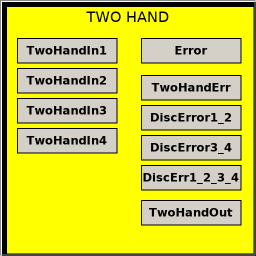
VISUALIZATION V_PH_TWOHAND  // 256x256
VAR_INPUT
	stSafetyTWOHAND			:ST_SAFETY_FBTWOHAND;
END_VAR
    Rectangle (2,2 256x256), colour toggle: stSafetyTWOHAND.bGeneralError
    Label (5,6 246x22), "TWO HAND"
    RoundedRectangle (17,38 100x25), "TwoHandIn1", colour toggle: stSafetyTWOHAND.uStatus.stStatusWords.wInputs.8
    RoundedRectangle (17,98 100x25), "TwoHandIn3", colour toggle: stSafetyTWOHAND.uStatus.stStatusWords.wInputs.10
    RoundedRectangle (17,68 100x25), "TwoHandIn2", colour toggle: stSafetyTWOHAND.uStatus.stStatusWords.wInputs.9
    RoundedRectangle (17,128 100x25), "TwoHandIn4", colour toggle: stSafetyTWOHAND.uStatus.stStatusWords.wInputs.11
    RoundedRectangle (141,38 100x25), "Error", colour toggle: stSafetyTWOHAND.uStatus.stStatusWords.wOutputs.0
    RoundedRectangle (141,200 100x25), "TwoHandOut", colour toggle: stSafetyTWOHAND.uStatus.stStatusWords.wOutputs.1
    RoundedRectangle (141,105 100x25), "DiscError1_2", colour toggle: stSafetyTWOHAND.uStatus.stStatusWords.wDiagnosis.0, invisible if: NOT stSafetyTWOHAND.uStatus.stStatusWords.wDiagnosis.0
    RoundedRectangle (141,75 100x25), "TwoHandErr", colour toggle: stSafetyTWOHAND.uStatus.stStatusWords.wDiagnosis.6
    RoundedRectangle (141,165 100x25), "DiscErr1_2_3_4", colour toggle: stSafetyTWOHAND.uStatus.stStatusWords.wDiagnosis.2, invisible if: NOT stSafetyTWOHAND.uStatus.stStatusWords.wDiagnosis.2
    RoundedRectangle (141,135 100x25), "DiscError3_4", colour toggle: stSafetyTWOHAND.uStatus.stStatusWords.wDiagnosis.1, invisible if: NOT stSafetyTWOHAND.uStatus.stStatusWords.wDiagnosis.1
    Textfield (17,226 234x25), text list: 'TL_FbState', text index: stSafetyTWOHAND.eState
END_VISUALIZATION

(* stored: Version 1.1.0.1, ProductVersion 3.1.4024.4
   Visu V_PH_TWOHAND: Id {a3e569b9-44b6-4440-8389-ee66fe1f7297} *)
